PROGRAM MAIN
VAR
	bShouldCalculate : BOOL;
	aDistances : ARRAY[1..24] OF INT;
	nStartPosition : INT := 1;
	nEndPosition: INT := 2;
	i: INT;
END_VAR

IF bShouldCalculate THEN
	FOR i := 1 TO 24 DO
		GLOBALS.aRoadFlags[i] := FALSE;
	END_FOR
	aDistances := DIJKSTRA(GLOBALS.stGraph, nStartPosition, nEndPosition);
	bShouldCalculate := FALSE;
END_IF

END_PROGRAM

(* stored: Version 1.1.0.1, ProductVersion 3.1.4024.12
   POU MAIN: Id {0a437958-698d-422f-9c03-3af28897c590}, SpecialFunc None *)
